FUNCTION switchWaterVentil : BOOL
VAR_INPUT
	bOpen : BOOL; // TRUE = öffnen, FALSE = schließen
	pMachine : POINTER TO FB_StateMachine;
END_VAR

IF (bOpen) THEN
	LogMessage(E_LogType.INFO, 'Betätige Ventil: -> ', 'öffnen');
ELSE
	LogMessage(E_LogType.INFO, 'Betätige Ventil: -> ', 'schliessen');
END_IF;	

IF bOpen THEN
	pMachine^.pd.actor.openFlowVentil := TRUE;
	pMachine^.pd.actor.closeFlowVentil := FALSE;
ELSE
	pMachine^.pd.actor.openFlowVentil := FALSE;
	pMachine^.pd.actor.closeFlowVentil := TRUE;
END_IF

END_FUNCTION

(* stored: Version 1.1.0.1
   POU switchWaterVentil: Id {2bfeaffd-a66e-4330-bc82-06133f12c6f8}, SpecialFunc None *)
